FUNCTION_BLOCK FB_LoadCell_SwomoConfig EXTENDS FB_ModbusSlaveRtu
VAR
	wAddRead : WORD;
	wAddWrite : WORD;
	wWriteLow : WORD;
	wWriteHigh : WORD;
	TmpData : TC3_Utilities_C.U_Word2Dint;
END_VAR

arrAddressRead[0][0] := wAddRead;
arrAddressRead[0][1] := 2;
arrAddressRead[0][2] := TC_ModbusBase.E_ModbusFunction.ReadHoldingRegisters;
iNumAddRegionRead := 1;

arrAddressWrite[0][0] := wAddWrite;
arrAddressWrite[0][1] := 2;
arrAddressWrite[0][2] := wWriteHigh;
arrAddressWrite[0][3] := wWriteLow;
arrAddressWrite[0][10] := E_ModbusFunction.WriteMultipleRegisters;

PROPERTY AddRead : WORD
GET
END_GET
SET
END_SET
END_PROPERTY

PROPERTY AddWrite : WORD
GET
END_GET
SET
END_SET
END_PROPERTY

METHOD Convert : BOOL
VAR_INPUT
	iRegionNo	: 	INT;
	pReadData	:	POINTER TO word;
END_VAR
CASE iRegionNo OF
	0:
		TmpData.iWord[1] := pReadData[0];
		TmpData.iWord[0] := pReadData[1];
END_CASE
END_METHOD

METHOD FirstCycle // must be call once time 
VAR_INPUT
	sName : STRING;
	iUnitID : BYTE ; // modbus address of the device : 1- 255
END_VAR
THIS^.sName := sName;
THIS^.iUnitID := iUnitID;
END_METHOD

PROPERTY WordWriteH : WORD
GET
END_GET
SET
END_SET
END_PROPERTY

PROPERTY WordWriteL : WORD
GET
END_GET
SET
END_SET
END_PROPERTY

END_FUNCTION_BLOCK

(* stored: Version 1.1.0.1, ProductVersion 3.1.4024.12
   POU FB_LoadCell_SwomoConfig: Id {1d1c2917-2e33-49d0-a8a4-f9fc8b2b5a9f}, SpecialFunc None
   Property AddRead: Id {d721851a-a112-4e3b-a313-8c38b9af5752}
   Get Get: Id {34b9d543-7766-4986-8c13-b18047169b65}
   Set Set: Id {ca46ddd0-ec40-4e12-95ec-277ee6fe8c80}
   Property AddWrite: Id {4aca9a36-4f11-4635-9be4-95dff1330437}
   Get Get: Id {df9940da-ba82-4ea9-a83f-a7b7cddf587a}
   Set Set: Id {48a7beff-b4e0-4f0e-9d2a-8a925f85834f}
   Method Convert: Id {fd1c70aa-b9b6-4bc1-8b81-6051f9f359a0}
   Method FirstCycle: Id {8ee8d0b9-38e0-40eb-96ec-fe04c6a68b42}
   Property WordWriteH: Id {d8244fe1-3321-48ab-99bc-b980b2731908}
   Get Get: Id {289947c2-66df-46bd-97fe-d0008ce66d05}
   Set Set: Id {d81efe65-d68a-4b6a-be65-525a6f52427f}
   Property WordWriteL: Id {a4adb634-ee7c-4510-988d-54e502878505}
   Get Get: Id {29524662-3df3-4918-8d51-fa4b5bb725b8}
   Set Set: Id {7ec7a558-ee4a-4c1d-a76f-e4a1f9bdc4b8} *)
